PROGRAM commandDecoder
VAR
	command 	: STRING(255);
	Head_Loaded : STRING;
	index 		: INT := 0;
	
	actualX 	: LREAL;
	actualY 	: LREAL;
	actualZ 	: Lreal;
	
	wait100ms : TON;
	
END_VAR

command := GVL.stReceivedData;
command := F_ToLCase(command);
GVL.stReceivedData := '';

wait100ms(IN := COM.bEnable, pt := T#500MS);

CASE index OF
	0:	//commands
		COM.bEnable := FALSE;
		COM.bCouple := FALSE;
		COM.bHome 	:= FALSE;
		COM.inUSe 	:= FALSE;
		
		IF 		(command = 'reset') THEN
			index := 10;
			command := '';
    	ELSIF 	(command = 'homing') THEN
			index := 100;
			command := '';
		ELSIF 	(command = 'z to zero') THEN
			index := 110;
			command := '';
		ELSIF 	(command = 'set vel') THEN
			index := 120;
			command := '';
		ELSIF 	(command = 'go xyz') THEN
			index := 200;
			command := '';
		ELSIF 	(command = 'go x') THEN
			index := 210;
			command := '';
		ELSIF 	(command = 'go y') THEN
			index := 220;
			command := '';
		ELSIF 	(command = 'go z') THEN
			index := 230;
			command := '';
		ELSIF 	(command = 'exec gcode') THEN
			index := 250;
			command := '';
		ELSIF 	(command = 'read pos') THEN
			index := 300;
			command := '';
		ELSIF 	(command = 'error') THEN
			index := 999;
			command := '';
		ELSE
			index := 0;
		END_IF;
		
	10: //reset
		COM.bReset 	:= TRUE;
		COM.bReset 	:= FALSE;
		
		COM.bEnable := FALSE;
		COM.bCouple := FALSE;
		COM.bHome 	:= FALSE;
		COM.inUSe 	:= FALSE;
		COM.bMoveX 	:= FALSE;
		COM.bMoveY 	:= FALSE;
		COM.bMoveZ 	:= FALSE;
		
		index 		:= 0;
		
	100: //Homing
		COM.bEnable := TRUE;
		COM.bCouple := TRUE;
		COM.bHome 	:= TRUE;
		
		IF COM.bHomeBusy THEN
			COM.inUSe 	:= TRUE;
		ELSE
			COM.inUSe 	:= FALSE;
		END_IF
		
		IF COM.bHomeDone THEN
			COM.bEnable := FALSE;
			COM.bCouple := FALSE;
			COM.bHome 	:= FALSE;
			COM.inUSe 	:= FALSE;
			index 	:= 0;
		END_IF
		
	110: //set Z position to zero
			COM.bSetZ 		:= TRUE;
			IF (COM.PosZ = 0 AND COM.bValid) THEN
				COM.bSetZ 	:= FALSE;
				index 		:= 0;
			END_IF
			
	120: //Set velocity
		COM.velX := 200;
		COM.velY := 200;
		COM.velZ := 2;
		index 		:= 0;
	
	200: //Go to xyz Pos
    	COM.absX := 100;
		COM.absY := 100;
		COM.absZ := 0;
		
		COM.bEnable := TRUE;
		COM.bCouple := TRUE;
		
		IF wait100ms.Q THEN 
			COM.bMoveX 	:= TRUE;
			COM.bMoveY 	:= TRUE;
			COM.bMoveZ 	:= TRUE;
		END_IF
		
		IF COM.bHomeBusy THEN
			COM.inUSe 	:= TRUE;
		ELSE
			COM.inUSe 	:= FALSE;
		END_IF
		
		IF COM.bMoveDone THEN
			COM.bEnable := FALSE;
			COM.bCouple := FALSE;
			COM.inUSe 	:= FALSE;
			COM.bMoveX 	:= FALSE;
			COM.bMoveY 	:= FALSE;
			COM.bMoveZ 	:= FALSE;
			index 	:= 0;
		END_IF
		
	210: //Go X Pos
	    COM.absX := 50;
		COM.bEnable := TRUE;
		COM.bCouple := TRUE;
		
		IF wait100ms.Q THEN 
			COM.bMoveX 	:= TRUE;
		END_IF
		
		IF COM.bHomeBusy THEN
			COM.inUSe 	:= TRUE;
		ELSE
			COM.inUSe 	:= FALSE;
		END_IF
		
		IF COM.bMoveXDone THEN
			COM.bEnable := FALSE;
			COM.bCouple := FALSE;
			COM.inUSe 	:= FALSE;
			COM.bMoveX 	:= FALSE;
			index 	:= 0;
		END_IF

	220: //Go Y Pos
		COM.bEnable := TRUE;
		COM.absY := 50;
		
		IF wait100ms.Q THEN 
			COM.bMoveY 	:= TRUE;
		END_IF
				
		IF COM.bHomeBusy THEN
			COM.inUSe 	:= TRUE;
		ELSE
			COM.inUSe 	:= FALSE;
		END_IF
		
		IF COM.bMoveYDone THEN
			COM.bEnable := FALSE;
			COM.bCouple := FALSE;
			COM.inUSe 	:= FALSE;
			COM.bMoveY 	:= FALSE;
			index 	:= 0;
		END_IF

	230: //Go Z Pos
		COM.absZ := -1;
		COM.bEnable := TRUE;
		
		IF wait100ms.Q THEN 
			COM.bMoveZ 	:= TRUE;
		END_IF
		
		IF COM.bHomeBusy THEN
			COM.inUSe 	:= TRUE;
		ELSE
			COM.inUSe 	:= FALSE;
		END_IF
		
		IF COM.bMoveZDone THEN
			COM.bEnable := FALSE;
			COM.bCouple := FALSE;
			COM.inUSe 	:= FALSE;
			COM.bMoveZ 	:= FALSE;
			index 	:= 0;
		END_IF
		
	250: //Execute Gcode--------------------------------------------------------------------------------------------
		
	300: //Read XYZ
		actualX 	:= COM.PosX;
		actualY 	:= COM.Posy;
		actualZ 	:= COM.PosZ;
		IF COM.bValid THEN
			index 	:= 0;
		END_IF

	999: //error
			COM.bEnable := FALSE;
			IF(command = 'reset')THEN
				index := 0;
			END_IF

	ELSE //errorstate
	index := 0;
END_CASE;

END_PROGRAM

(* stored: Version 1.1.0.1, ProductVersion 3.1.4024.2
   POU commandDecoder: Id {7eba7217-46bb-46ef-8690-bb184ce360f6}, SpecialFunc None *)
